//
// This FB calculates resulting pressure applying the selected voting method.
// Up to five pressure sensors are used in the calculation.
// The resulting value is a combination of values from available/valid sensors.
// For more info, see method M_SetStatus().
//
FUNCTION_BLOCK FB_CRYO_PRESSURE_VOTE
VAR_INPUT
	{attribute 'OPC.UA.DA' := '0'}
	in_bSimulation:	BOOL	:= FALSE;	// If TRUE, the pressure value is simulated.
	
	{attribute 'OPC.UA.DA' := '0'}
	in_nNumSensor:	INT;				// Number of sensors used by voiting method.
	
	{attribute 'OPC.UA.DA' := '0'}
	in_nVoteMethod:	E_CRYO_VOTE	:= E_CRYO_VOTE.V_AVE;	// Active voting method.
	
	// Five pointers to instances of FB_CRYO_SENSOR_PRESSURE.
	// Pointers should only be set to existing pressure sensors.
	{attribute 'OPC.UA.DA' := '0'}
	in_pSensor1:		POINTER TO FB_CRYO_SENSOR_PRESSURE	:= 0;
	{attribute 'OPC.UA.DA' := '0'}
	in_pSensor2:		POINTER TO FB_CRYO_SENSOR_PRESSURE	:= 0;
	{attribute 'OPC.UA.DA' := '0'}
	in_pSensor3:		POINTER TO FB_CRYO_SENSOR_PRESSURE	:= 0;
	{attribute 'OPC.UA.DA' := '0'}
	in_pSensor4:		POINTER TO FB_CRYO_SENSOR_PRESSURE	:= 0;
	{attribute 'OPC.UA.DA' := '0'}
	in_pSensor5:		POINTER TO FB_CRYO_SENSOR_PRESSURE	:= 0;

END_VAR
VAR
	{attribute 'OPC.UA.DA' := '1'}
	stat:		T_CRYO_PRESSURE_VOTE_STATUS;	// Complete status
	
	pSensor:	ARRAY [1..5] OF POINTER TO FB_CRYO_SENSOR_PRESSURE;
END_VAR

// If not configured yet, return.
IF NOT M_Configure()	THEN
	RETURN;
END_IF

// Set warnings for sensors with problems
M_CheckWarnings();

// Set the calculated vacuum pressure
M_SetStatus();

METHOD M_CheckWarnings : BOOL
VAR_INPUT
END_VAR
VAR
	i:			INT;
END_VAR
FOR i:=1 TO in_nNumSensor DO
	IF pSensor[i] <> 0  THEN
		// The set pointer (<> 0) indicates that the sensor is connected.
		// Warnings could be set only for connected sensors.
		IF  pSensor[i]^.stat.bValid	THEN
			// Clear warning
			M_SetWarning(i, FALSE);
		ELSE
			// Set warning
			M_SetWarning(i, TRUE);
		END_IF
	ELSE
		// Not connected sensors don't have warnings
		M_SetWarning(i, FALSE);
	END_IF
END_FOR
END_METHOD

METHOD M_Configure : BOOL
VAR_INPUT
END_VAR
VAR
	j:					INT;
END_VAR
VAR_INST
	{attribute 'OPC.UA.DA' := '0'}
	i:	INT := 0;
	{attribute 'OPC.UA.DA' := '0'}
	bConfigured:	BOOL := FALSE;
END_VAR
// The number of sensors must be between 1 and 5.
IF in_nNumSensor < 1 OR in_nNumSensor > 5 THEN
	// Set error string
	stat.sStatus	:= 'ERROR: Number of sensors (var in_nNumSensor) is not in range [1..5]';
	RETURN;
END_IF

// Configure the system in stages after boot-up.
// WARNING:
// It seems that setting of pointers takes some time and cannot be done in FB_Init.
// After 40 cycles, we set pointers to sensors.
// After 80 cycles, we set general configuration parameters and complete configuration.
IF NOT bConfigured THEN
	i	:= i + 1;
	IF i = 40 THEN
		// Assign pointers to the sensor device instances
		pSensor[1] := in_pSensor1;
		pSensor[2] := in_pSensor2;
		pSensor[3] := in_pSensor3;
		pSensor[4] := in_pSensor4;
		pSensor[5] := in_pSensor5;
	ELSIF i >= 80 THEN
		FOR j := 1 TO in_nNumSensor DO
			IF pSensor[j] <> 0 THEN
				// Set the status flag that the sensor is connected.
				M_SetConnected(j, TRUE);
				// At least one pointer is not zero.
				// We have finished configuration.
				bConfigured	:= TRUE;
			ELSE
				M_SetConnected(j, FALSE);
			END_IF
		END_FOR
	END_IF
END_IF

M_Configure	:= bConfigured;
END_METHOD

METHOD M_SetConnected : BOOL
VAR_INPUT
	in_nIndex:		INT;
	in_bConnected:	BOOL;
END_VAR
CASE in_nIndex OF
	1:
		stat.bConnSens1	:= in_bConnected;
	2:
		stat.bConnSens2	:= in_bConnected;
	3:
		stat.bConnSens3	:= in_bConnected;
	4:
		stat.bConnSens4	:= in_bConnected;
	5:
		stat.bConnSens5	:= in_bConnected;
END_CASE
END_METHOD

// Calculate pressure based on the status of the two sensors
METHOD M_SetStatus
VAR_INPUT
END_VAR
VAR
	lrTmp:		LREAL;	// Temporary var
	nSample:	INT;
	i:			INT;
END_VAR
//
// If simulated, set the simulated value and return.
//
IF in_bSimulation THEN
	stat.bSimulated	:= TRUE;
	stat.bValid		:= TRUE;
	stat.lrPressure	:= stat.lrSimPressure;
	RETURN;
ELSE
	stat.bSimulated	:= FALSE;
END_IF


//
// Get the pressure depending on the voting method.
//
CASE in_nVoteMethod OF
	E_CRYO_VOTE.V_AVE:
		M_SetStatus_Average();
	E_CRYO_VOTE.V_MIN:
		M_SetStatus_Minimum();
	E_CRYO_VOTE.V_MAX:
		M_SetStatus_Maximum();
	E_CRYO_VOTE.V_1oo2:
		M_SetStatus_FirstValid();
	E_CRYO_VOTE.V_2oo3:
		M_SetStatus_XooY(2,3);
	E_CRYO_VOTE.V_3oo5:
		M_SetStatus_XooY(3,5);
ELSE
	;
END_CASE


//
// If the reading is valid, set the simulated value to it.
// This way, switching from normal to simulation will result in
// no jump in the value.
//
IF stat.bValid  THEN
	stat.lrSimPressure	:= stat.lrPressure;
END_IF
END_METHOD

// Calculate pressure based on the average of all valid sensor readings
METHOD M_SetStatus_Average
VAR_INPUT
END_VAR
VAR
	lrTmp:		LREAL;	// Temporary var for sum of pressures
	nSample:	INT;	// Number of valid sensor readings
	i:			INT;
END_VAR
lrTmp	:= 0.0;
nSample	:= 0;
FOR i:=1 TO in_nNumSensor DO
	IF pSensor[i] <> 0  THEN
		IF  pSensor[i]^.stat.bValid	THEN
			lrTmp	:= lrTmp + pSensor[i]^.stat.lrPressure;
			nSample	:= nSample + 1;
		END_IF
	END_IF
END_FOR
IF nSample > 0	THEN
	stat.lrPressure	:= lrTmp / nSample;
	stat.bValid		:= TRUE;
ELSE
	stat.lrPressure	:= 9999;
	stat.bValid		:= FALSE;
END_IF
END_METHOD

// Calculate pressure based on the first measured valid value
METHOD M_SetStatus_FirstValid
VAR_INPUT
END_VAR
VAR
	lrTmp:		LREAL;	// Temporary var for sum of pressures
	nSample:	INT;	// Number of valid sensor readings
	i:			INT;
END_VAR
nSample	:= 0;
FOR i:=1 TO in_nNumSensor DO
	IF pSensor[i] <> 0  THEN
		IF  pSensor[i]^.stat.bValid	THEN
			lrTmp	:= pSensor[i]^.stat.lrPressure;
			nSample	:= nSample + 1;
			EXIT;
		END_IF
	END_IF
END_FOR
IF nSample > 0	THEN
	stat.lrPressure	:= lrTmp;
	stat.bValid		:= TRUE;
ELSE
	stat.lrPressure	:= 9999;
	stat.bValid		:= FALSE;
END_IF
END_METHOD

// Calculate pressure based on the highest measured valid value
METHOD M_SetStatus_Maximum
VAR_INPUT
END_VAR
VAR
	lrTmp:		LREAL;	// Temporary var for sum of pressures
	nSample:	INT;	// Number of valid sensor readings
	i:			INT;
END_VAR
lrTmp	:= -100000.0;	// Dummy starting value
nSample	:= 0;
FOR i:=1 TO in_nNumSensor DO
	IF pSensor[i] <> 0  THEN
		IF  pSensor[i]^.stat.bValid	THEN
			IF pSensor[i]^.stat.lrPressure > lrTmp THEN
				lrTmp	:= pSensor[i]^.stat.lrPressure;
			END_IF
			nSample	:= nSample + 1;
		END_IF
	END_IF
END_FOR
IF nSample > 0	THEN
	stat.lrPressure	:= lrTmp;
	stat.bValid		:= TRUE;
ELSE
	stat.lrPressure	:= 9999;
	stat.bValid		:= FALSE;
END_IF
END_METHOD

// Calculate pressure based on the lowest measured valid value
METHOD M_SetStatus_Minimum
VAR_INPUT
END_VAR
VAR
	lrTmp:		LREAL;	// Temporary var for sum of pressures
	nSample:	INT;	// Number of valid sensor readings
	i:			INT;
END_VAR
lrTmp	:= 100000.0;	// Dummy starting value
nSample	:= 0;
FOR i:=1 TO in_nNumSensor DO
	IF pSensor[i] <> 0  THEN
		IF  pSensor[i]^.stat.bValid	THEN
			IF pSensor[i]^.stat.lrPressure < lrTmp THEN
				lrTmp	:= pSensor[i]^.stat.lrPressure;
			END_IF
			nSample	:= nSample + 1;
		END_IF
	END_IF
END_FOR
IF nSample > 0	THEN
	stat.lrPressure	:= lrTmp;
	stat.bValid		:= TRUE;
ELSE
	stat.lrPressure	:= 9999;
	stat.bValid		:= FALSE;
END_IF
END_METHOD

// Calculate pressure based on the status of the two sensors
METHOD M_SetStatus_XooY
VAR_INPUT
	in_nNum:	INT;	// Number of readings to select for voting (X)
	in_nTotal:	INT;	// Total number of readings to check (Y)
END_VAR
VAR
	idx_i, idx_j:	INT;
	nTmp:		INT;			// Temporary INT var
	lrTmp:		LREAL	:= 0.0;	// Temporary var for sum of pressures
	nValid:		INT		:= 0;	// Total number of valid readings
	nSample:	INT		:= 0;	// Number of valid sensor readings
	
	aDiff:		ARRAY [1..5,1..5] OF LREAL;	// Table of absolute differences
	aDiffSum:	ARRAY [1..5] OF LREAL;		// Array of sums of absolute differences
	// Array of indexes of sums of absolute differences
	aDiffSumIdx:ARRAY [1..5] OF INT := [1,2,3,4,5];		
	lrAbsDiff:	LREAL;						// Absolute difference between two readings
	
	i:			INT;
	j:			INT;
END_VAR
//
//	Get the number of valid readings and calculate the average
//
FOR i:=1 TO in_nTotal DO
	IF pSensor[i] <> 0  THEN
		IF  pSensor[i]^.stat.bValid	THEN
			lrTmp	:= lrTmp + pSensor[i]^.stat.lrPressure;
			nValid	:= nValid + 1;
		END_IF
	END_IF
END_FOR


//
// Vote X out of Y
//
IF nValid >= in_nNum	THEN
	//
	// Calculate relative differences between two readings, 
	// relative to the bigger ABS value.
	// Table is symetric. Calculate only the half (triangle) on the right. 
	// Make a copy to the other half.
	//
	FOR i:=1 TO in_nTotal DO
		FOR j:=i+1 TO in_nTotal DO
			IF pSensor[i] <> 0  AND  pSensor[j] <> 0	THEN
				IF pSensor[i]^.stat.bValid  AND  pSensor[j]^.stat.bValid	THEN
					lrAbsDiff	:= ABS(pSensor[i]^.stat.lrPressure - pSensor[j]^.stat.lrPressure);
					aDiff[i,j]	:= lrAbsDiff;
					aDiff[j,i]	:= lrAbsDiff;
				ELSE
					aDiff[i,j]	:= 9999.0;
					aDiff[j,i]	:= 9999.0;
				END_IF
			ELSE
				aDiff[i,j]	:= 9999.0;
				aDiff[j,i]	:= 9999.0;
			END_IF
		END_FOR
	END_FOR

	//
	// Get the sum of all differences for each reading.
	//
	FOR i:=1 TO in_nTotal DO
		aDiffSum[i]	:= 0.0;
		FOR j:=1 TO in_nTotal DO
			aDiffSum[i]	:= aDiffSum[i] + aDiff[i,j];
		END_FOR
	END_FOR

	//
	// Sort the indexes for differences in accending order (low sum first).
	//
	FOR i:=1 TO in_nTotal DO
		FOR j:=i+1 TO in_nTotal DO
			idx_i	:= aDiffSumIdx[i];
			idx_j	:= aDiffSumIdx[j];
			IF aDiffSum[idx_j] < aDiffSum[idx_i]	THEN
				// Swap indexes
				nTmp			:= aDiffSumIdx[j];
				aDiffSumIdx[j]	:= aDiffSumIdx[i];
				aDiffSumIdx[i]	:= nTmp;
			END_IF
		END_FOR
	END_FOR

	
	//					
	// Get the average of selected in_nNum readings.
	// Assign the result to the pressure.
	//
	lrTmp	:= 0.0;
	FOR i:=1 TO in_nNum DO
		idx_i	:= aDiffSumIdx[i];
		lrTmp	:= lrTmp + pSensor[idx_i]^.stat.lrPressure;
	END_FOR
	
	stat.lrPressure	:= lrTmp / in_nNum;
	stat.bValid		:= TRUE;
ELSE
	stat.lrPressure	:= 9999;
	stat.bValid		:= FALSE;
END_IF
END_METHOD

METHOD M_SetWarning : BOOL
VAR_INPUT
	in_nIndex:		INT;
	in_bWarning:	BOOL;
END_VAR
CASE in_nIndex OF
	1:
		stat.bWarnSens1	:= in_bWarning;
	2:
		stat.bWarnSens2	:= in_bWarning;
	3:
		stat.bWarnSens3	:= in_bWarning;
	4:
		stat.bWarnSens4	:= in_bWarning;
	5:
		stat.bWarnSens5	:= in_bWarning;
END_CASE
END_METHOD

END_FUNCTION_BLOCK

(* stored: Version 1.1.0.1, ProductVersion 3.1.4024.12
   POU FB_CRYO_PRESSURE_VOTE: Id {a9baf80f-f196-4114-847c-ebe5cf64e1c7}, SpecialFunc None
   Method M_CheckWarnings: Id {97ccceae-71ae-4edf-a5e3-56878805dcf6}
   Method M_Configure: Id {899f2132-8105-4993-a4e7-0e233b23a383}
   Method M_SetConnected: Id {0385cbd9-0a92-4fea-89c9-aad633d40dc0}
   Method M_SetStatus: Id {50c6dbc8-aee5-4d9b-9594-29f858321371}
   Method M_SetStatus_Average: Id {f663c67c-9fa1-4932-8abb-f049d4f62c65}
   Method M_SetStatus_FirstValid: Id {fc557b5a-1c63-4a2c-bcd9-e603834a10ed}
   Method M_SetStatus_Maximum: Id {7eb7fe8f-29c1-4676-8d32-dd71cea6b81a}
   Method M_SetStatus_Minimum: Id {60bee11a-9d21-4da8-8f27-86d24ca49a88}
   Method M_SetStatus_XooY: Id {1582a26d-963f-4ead-8699-e31d58d514a7}
   Method M_SetWarning: Id {349817fc-01ba-4490-a7e4-2e8d5056a0a7} *)
